{attribute 'linkalways'} 
{attribute 'no_explicit_call' := 'This FB is a CLASS and must be accessed using methods or properties'}
{attribute 'enable_dynamic_creation'}
FUNCTION_BLOCK _ETcVnDistanceTransformationLabel EXTENDS EnumDatatypeBase
VAR
	localData : ETcVnDistanceTransformationLabel;
	activeData : REFERENCE TO ETcVnDistanceTransformationLabel;
	enumBaseDatatype : _DINT(localData);
END_VAR

METHOD PRIVATE AddLocalEnumeration
VAR_INPUT
	Enumeration : T_MAXSTRING;
	Value : ETcVnDistanceTransformationLabel;
END_VAR
AddEnumeration(Enumeration, Value);
END_METHOD

PROPERTY PUBLIC Address : PVOID
GET
Address := ADR(activeData);
END_GET
END_PROPERTY

METHOD PUBLIC ClearReference
VAR_INPUT
END_VAR
activeData REF= localData;
SetBaseDatatypeReference();
END_METHOD

METHOD PUBLIC Clone : I_Datatype
VAR
    pClone : POINTER TO _ETcVnDistanceTransformationLabel;
END_VAR
pClone := __NEW(_ETcVnDistanceTransformationLabel(InitialValue := Value));
Clone := pClone^;
END_METHOD

METHOD FB_init : BOOL
VAR_INPUT
	bInitRetains : BOOL; // if TRUE, the retain variables are initialized (warm start / cold start)
	bInCopyCode : BOOL;  // if TRUE, the instance afterwards gets moved into the copy code (online change)
	InitialValue : ETcVnDistanceTransformationLabel;
END_VAR
localData := InitialValue;
AddBaseDatatype(enumBaseDatatype);
ClearReference();

AddLocalEnumeration('TCVN_DTL_CCOMP', ETcVnDistanceTransformationLabel.TCVN_DTL_CCOMP);
AddLocalEnumeration('TCVN_DTL_PIXEL', ETcVnDistanceTransformationLabel.TCVN_DTL_PIXEL);
END_METHOD

PROPERTY PUBLIC Identifier : T_MAXSTRING
GET
Identifier := 'ETcVnDistanceTransformationLabel';
END_GET
END_PROPERTY

METHOD IsEnumeratorValueEqual : BOOL
VAR_INPUT
	Enumerator : I_KeyValueForwardEnumerator;
END_VAR
VAR
	storedValue : ETcVnDistanceTransformationLabel;
END_VAR
IF NOT Enumerator.TryGet(storedValue) THEN
	RETURN;
END_IF

IsEnumeratorValueEqual := storedValue = activeData;
END_METHOD

METHOD PUBLIC MakeReferenceTo
VAR_INPUT
	ReferenceTarget : REFERENCE TO ETcVnDistanceTransformationLabel;
END_VAR
activeData REF= ReferenceTarget;
SetBaseDatatypeReference();
END_METHOD

METHOD PROTECTED SetBaseDatatypeReference
VAR_INPUT
END_VAR
enumBaseDatatype.MakeReferenceTo(activeData);
END_METHOD

PROPERTY PUBLIC Size : UDINT
GET
Size := SIZEOF(activeData);
END_GET
END_PROPERTY

METHOD TryMakeReferenceTo : BOOL
VAR_INPUT
	Target : I_Datatype;
END_VAR
VAR
	targetAsEnum : I_EnumDatatype;
	pTargetData : POINTER TO ETcVnDistanceTransformationLabel;
END_VAR
IF NOT Target.TryResolveAsEnumDatatype(targetAsEnum) THEN
	RETURN;
END_IF

IF targetAsEnum.Identifier <> Identifier THEN
	RETURN;
END_IF

pTargetData := Target.Address;
activeData REF= pTargetData^;
SetBaseDatatypeReference();
TryMakeReferenceTo := TRUE;
END_METHOD

PROPERTY PUBLIC Value : ETcVnDistanceTransformationLabel
GET
Value := activeData;
END_GET
SET
activeData := Value;
END_SET
END_PROPERTY

END_FUNCTION_BLOCK

(* stored: Version 1.1.0.1, ProductVersion 3.1.4024.12
   POU _ETcVnDistanceTransformationLabel: Id {83a8242e-f6d1-4d46-8bfc-b3346e0665c0}, SpecialFunc None
   Folder Constructor: Id {47822503-8ec4-44ca-b6f9-7bdfae83aaa9}
   Folder Private: Id {e4133766-84fd-423a-b5b6-9d79f0475a25}
   Folder Protected: Id {32613942-bdac-4732-805c-58bea70b2e13}
   Method AddLocalEnumeration: Id {7e824379-4d55-47d1-92d0-58ce4bfba519}
   Property Address: Id {c9bdf049-97b2-472c-948e-c09cdc0f9318}
   Get Get: Id {27b0777d-63d7-4472-b1bf-cb4b4360d5da}
   Method ClearReference: Id {68834e4b-9101-47d4-8d2b-c0c3bb6d23dc}
   Method Clone: Id {1fa40b03-fff8-4598-8de8-b21213f95b8c}
   Method FB_init: Id {41c34a6c-f101-4af9-8e00-4223c750acf0}
   Property Identifier: Id {9c6c5756-8cbf-455e-a2e6-1208be3a2440}
   Get Get: Id {d430a535-49df-460d-b55a-27fdb41a85e5}
   Method IsEnumeratorValueEqual: Id {c5209143-8fec-4707-a85d-08c61aed5a35}
   Method MakeReferenceTo: Id {a3b558cd-d43b-44a8-9fbe-3c448fcc9cc1}
   Method SetBaseDatatypeReference: Id {8cc0e2f4-3f1a-4e56-bfcf-628203d0b42e}
   Property Size: Id {651fe06b-4566-4b16-a057-ff0ae007ca70}
   Get Get: Id {98feec80-d98e-4170-835a-cbb10855146e}
   Method TryMakeReferenceTo: Id {28b684e8-caa9-415d-916b-ea2dddbe8ca8}
   Property Value: Id {ac8c50fb-9a5a-407a-9239-1703155a924f}
   Get Get: Id {49cc06a4-2889-4922-b374-0bb7af652658}
   Set Set: Id {c6584432-a5a9-4817-84d3-3e200623363f} *)
